PROGRAM UnitTestProgram
VAR
	MotorControl_Test : FB_MotorControl_Test;
END_VAR

TcUnit.RUN();

END_PROGRAM

(* stored: Version 1.1.0.1, ProductVersion 3.1.4024.12
   POU UnitTestProgram: Id {6ee97de3-1527-4e60-9cef-4d70f0e42f35}, SpecialFunc None *)
